FUNCTION_BLOCK MotorControl IMPLEMENTS I_Motor
VAR
	OnOff AT%Q* : BOOL;
END_VAR

METHOD PUBLIC Start
VAR_INPUT
END_VAR
OnOff	:=	TRUE;
END_METHOD

METHOD PUBLIC stop : BOOL
VAR_INPUT
END_VAR
OnOff := FALSE;
END_METHOD

END_FUNCTION_BLOCK

(* stored: Version 1.1.0.1, ProductVersion 3.1.4024.12
   POU MotorControl: Id {5a51c125-03a7-4d40-a9ff-485e5602c3fb}, SpecialFunc None
   Method Start: Id {781b6612-0b89-49ea-af73-a8312f29dbf4}
   Method stop: Id {b2468803-54da-4f91-be8b-d8e603f4555e} *)
